PROGRAM PRG_ACTUATORS
VAR
END_VAR

MPA_321();
MPA_322();
MPA_323();
MPA_324();
MPA_325();
MPA_326();
MPA_327();
MPA_328();
MPA_329();

END_PROGRAM

(* stored: Version 1.1.0.1, ProductVersion 3.1.4022.16
   POU PRG_ACTUATORS: Id {2eccc79f-a12c-40ff-a593-4981b0ae670c}, SpecialFunc None *)
